Yaskawa INFORM job: READTWS_A.JBI

/JOB
//NAME READTWS_A
///FOLDERNAME MASTER
//POS
///NPOS 0,0,0,0,0,0
//INST
///DATE 2021/10/29 11:49
///ATTR SC,RO
NOP
'*****************************
'READ THE LEFT TWO DIGITS OF
'TWS AND SET IN B010.
'*****************************
DOUT OT#(17) OFF
DOUT OT#(18) OFF
DOUT OT#(19) ON
DOUT OT#(20) OFF
TIMER T=0.20
DIN B010 IGH#(5)
TIMER T=0.10
DOUT OT#(19) OFF
DOUT OT#(20) ON
TIMER T=0.20
DIN B011 IGH#(5)
TIMER T=0.10
DOUT OT#(20) OFF
MUL B011 10
ADD B010 B011
END
